% RSLogix 500 project CAR_PARKING_SYSTEM_BAK000.RSS, saved by version 8.30.00.16 %
PROJECT "UNTITLED"    % processor: Bul.1763 MicroLogix 1100 Series B %

PROGRAM FILES
  LAD 2   7 rungs

DATA FILES
  O0 OUTPUT  4 elements
  I1 INPUT  6 elements
  S2 STATUS  66 elements
  B3 BINARY  1 elements
  T4 TIMER  1 elements
  C5 COUNTER  1 elements
  R6 CONTROL  1 elements
  N7 INTEGER  1 elements
  F8 FLOAT  1 elements

LADDER 2
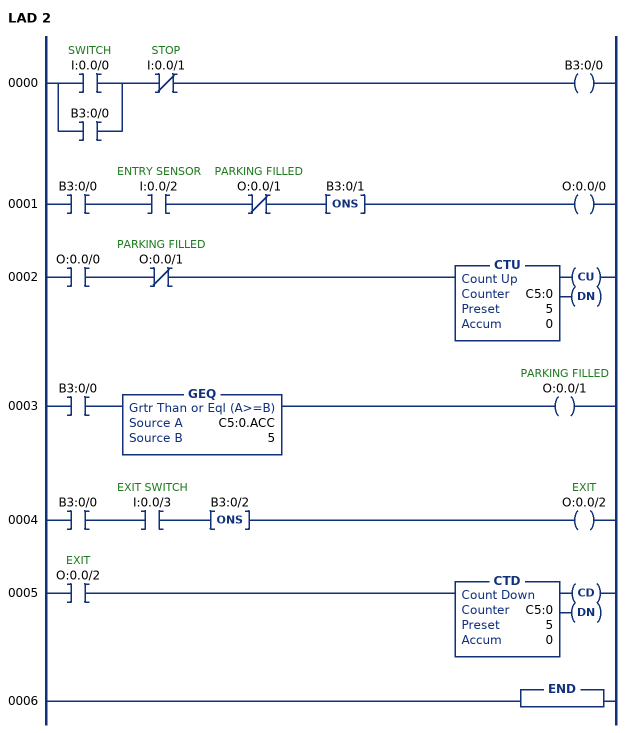
% Rung: 0 %
SOR BST XIC I:0.0/0 NXB XIC B3:0/0 BND XIO I:0.0/1 OTE B3:0/0 EOR
%   I:0.0/0  "SWITCH" %
%   I:0.0/1  "STOP" %
% Rung: 1 %
SOR XIC B3:0/0 XIC I:0.0/2 XIO O:0.0/1 ONS B3:0/1 OTE O:0.0/0 EOR
%   I:0.0/2  "ENTRY SENSOR" %
%   O:0.0/1  "PARKING FILLED" %
% Rung: 2 %
SOR XIC O:0.0/0 XIO O:0.0/1 CTU C5:0 5 0 EOR
%   O:0.0/1  "PARKING FILLED" %
% Rung: 3 %
SOR XIC B3:0/0 GEQ C5:0.ACC 5 OTE O:0.0/1 EOR
%   O:0.0/1  "PARKING FILLED" %
% Rung: 4 %
SOR XIC B3:0/0 XIC I:0.0/3 ONS B3:0/2 OTE O:0.0/2 EOR
%   I:0.0/3  "EXIT SWITCH" %
%   O:0.0/2  "EXIT" %
% Rung: 5 %
SOR XIC O:0.0/2 CTD C5:0 5 0 EOR
%   O:0.0/2  "EXIT" %
% Rung: 6 %
SOR END EOR

DATA TABLE (non-zero values as saved)
DATA C5
% .PRE .ACC %
% C5:0 % 5 0
